TYPE DUT :
STRUCT
END_STRUCT
END_TYPE

(* stored: Version 1.1.0.1, ProductVersion 3.1.4024.12
   DUT DUT: Id {2ad943d3-42df-4541-be61-bfdbaea57c4a} *)
